(* IEC 61131-3 sources: log21/plc-runtime/plc/edit_plc, 1 file *)

(* ---- prova.plc ---- *)
VAR_GLOBAL
	_CREATED : UDINT:= 1108581922;
	_VERSION : STRING:= '1.0.0.0';
END_VAR

PROGRAM NONAME
	LD	III
	ST	OOO

END_PROGRAM
